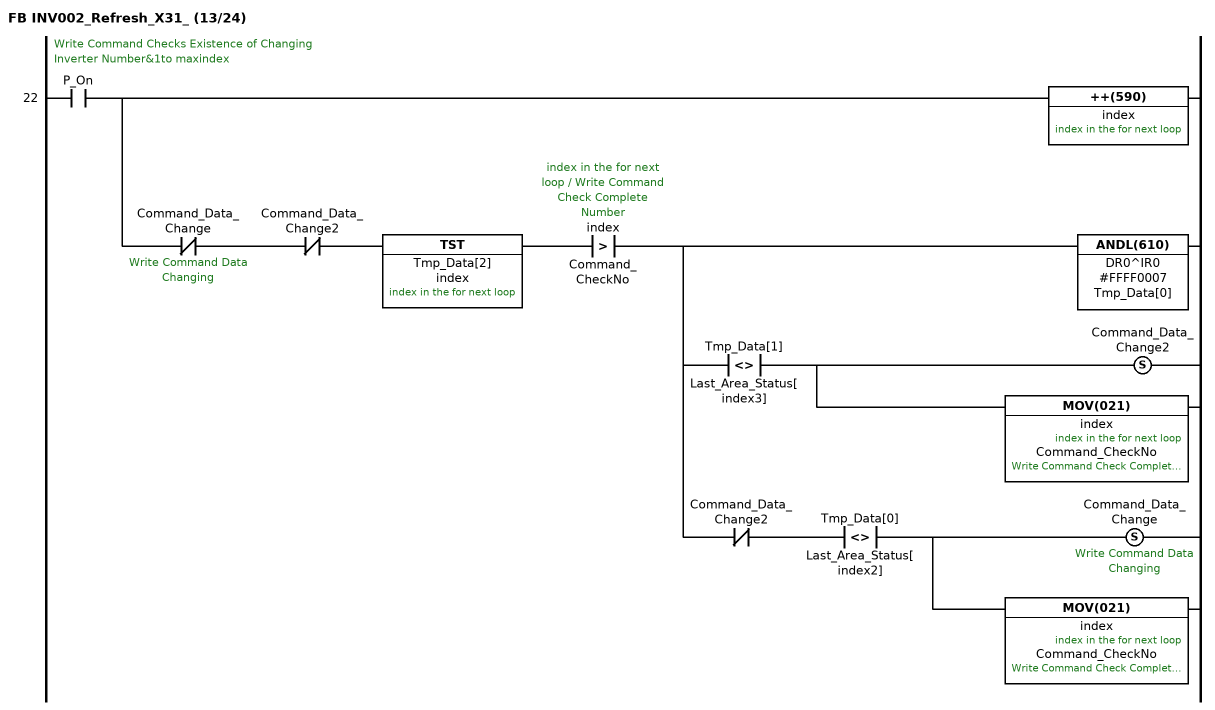
; [picture p24: FB INV002_Refresh_X31_, rungs 22-22]
; rung 22: Write Command Checks Existence of Changing / Inverter Number&1to maxindex
LD P_On
++(590) index  ; index in the for next loop
ANDNOT Command_Data_Change  ; Write Command Data Changing
ANDNOT Command_Data_Change2
ANDTST(350) Tmp_Data[2] index  ; index in the for next loop
AND>(320) index Command_CheckNo  ; index in the for next loop, Write Command Check Complete Number
OUT TR0
ANDL(610) DR0^IR0 #FFFF0007 Tmp_Data[0]
AND<>(305) Tmp_Data[1] Last_Area_Status[index3]
SET Command_Data_Change2
MOV(021) index Command_CheckNo  ; index in the for next loop, Write Command Check Complete Number
LD TR0
ANDNOT Command_Data_Change2
AND<>(305) Tmp_Data[0] Last_Area_Status[index2]
SET Command_Data_Change  ; Write Command Data Changing
MOV(021) index Command_CheckNo  ; index in the for next loop, Write Command Check Complete Number

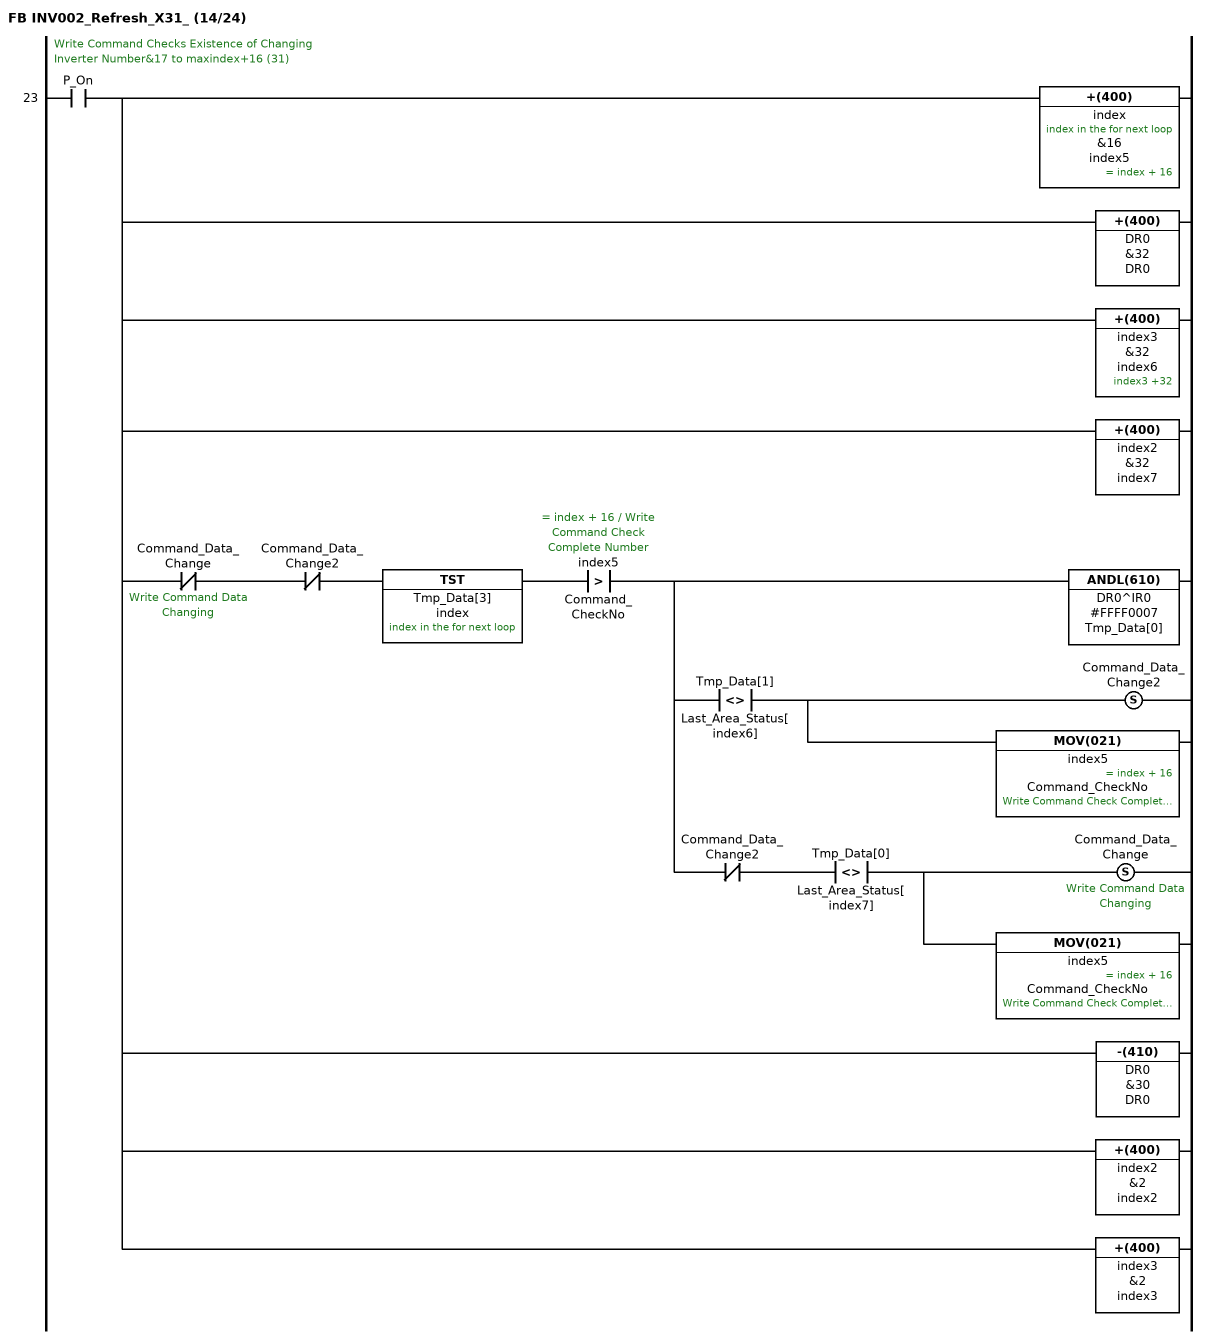
; rung 23: Write Command Checks Existence of Changing / Inverter Number&17 to maxindex+16 (31)
LD P_On
OUT TR0
+(400) index &16 index5  ; index in the for next loop, = index + 16
+(400) DR0 &32 DR0
+(400) index3 &32 index6  ; index3 +32
+(400) index2 &32 index7
ANDNOT Command_Data_Change  ; Write Command Data Changing
ANDNOT Command_Data_Change2
ANDTST(350) Tmp_Data[3] index  ; index in the for next loop
AND>(320) index5 Command_CheckNo  ; = index + 16, Write Command Check Complete Number
OUT TR1
ANDL(610) DR0^IR0 #FFFF0007 Tmp_Data[0]
AND<>(305) Tmp_Data[1] Last_Area_Status[index6]
SET Command_Data_Change2
MOV(021) index5 Command_CheckNo  ; = index + 16, Write Command Check Complete Number
LD TR1
ANDNOT Command_Data_Change2
AND<>(305) Tmp_Data[0] Last_Area_Status[index7]
SET Command_Data_Change  ; Write Command Data Changing
MOV(021) index5 Command_CheckNo  ; = index + 16, Write Command Check Complete Number
LD TR0
-(410) DR0 &30 DR0
+(400) index2 &2 index2
+(400) index3 &2 index3

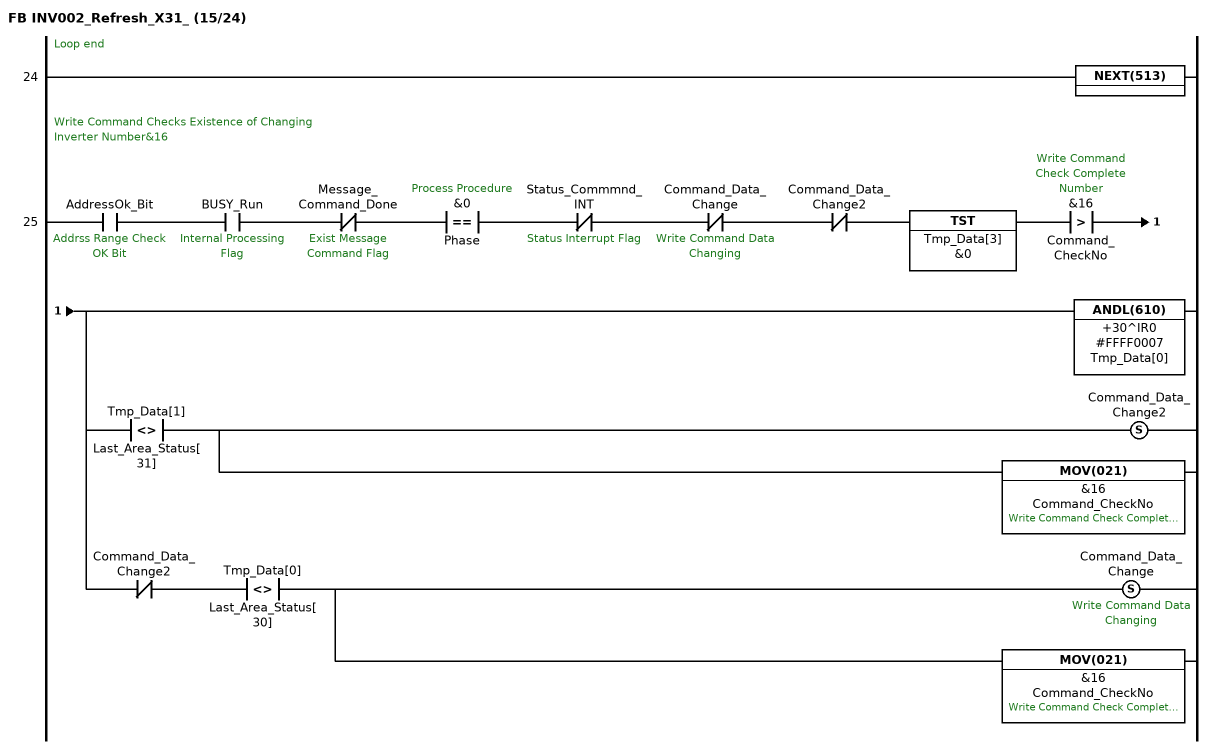
; rung 24: Loop end
NEXT(513)
; rung 25: Write Command Checks Existence of Changing / Inverter Number&16
LD AddressOk_Bit  ; Addrss Range Check OK Bit
AND BUSY_Run  ; Internal Processing Flag
ANDNOT Message_Command_Done  ; Exist Message Command Flag
AND=(300) &0 Phase  ; Process Procedure
ANDNOT Status_Commmnd_INT  ; Status Interrupt Flag
ANDNOT Command_Data_Change  ; Write Command Data Changing
ANDNOT Command_Data_Change2
ANDTST(350) Tmp_Data[3] &0
AND>(320) &16 Command_CheckNo  ; Write Command Check Complete Number
OUT TR0
ANDL(610) +30^IR0 #FFFF0007 Tmp_Data[0]
AND<>(305) Tmp_Data[1] Last_Area_Status[31]
SET Command_Data_Change2
MOV(021) &16 Command_CheckNo  ; Write Command Check Complete Number
LD TR0
ANDNOT Command_Data_Change2
AND<>(305) Tmp_Data[0] Last_Area_Status[30]
SET Command_Data_Change  ; Write Command Data Changing
MOV(021) &16 Command_CheckNo  ; Write Command Check Complete Number

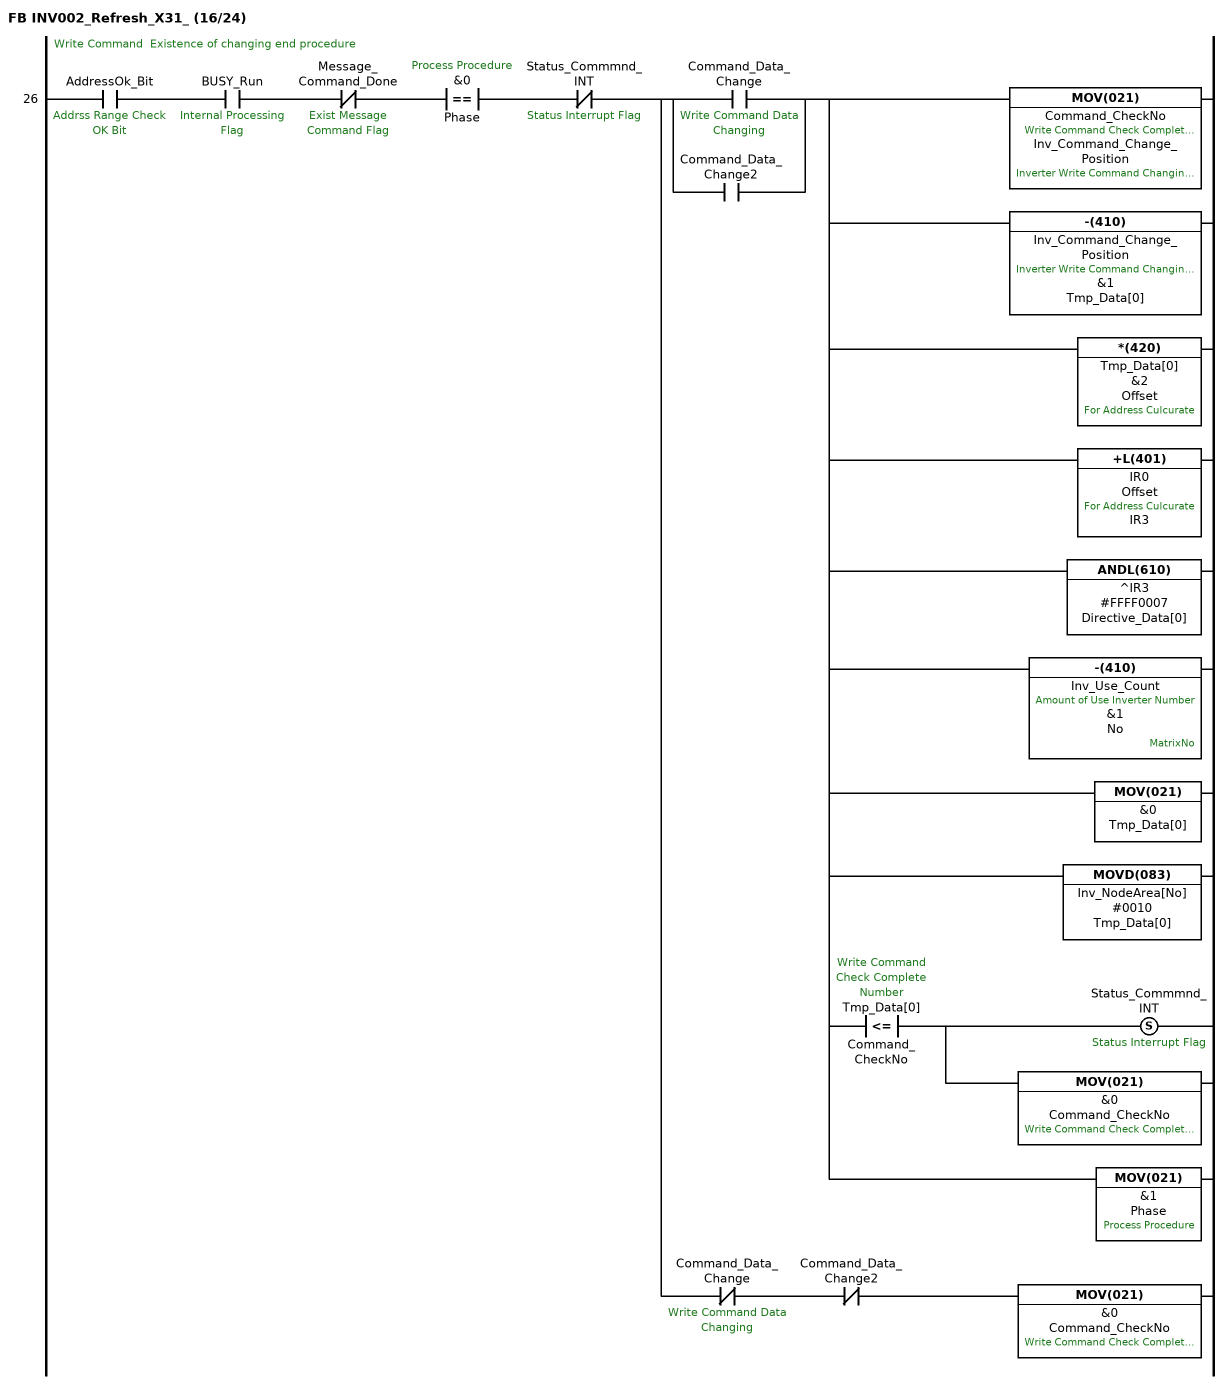
; rung 26: Write Command  Existence of changing end procedure
LD AddressOk_Bit  ; Addrss Range Check OK Bit
AND BUSY_Run  ; Internal Processing Flag
ANDNOT Message_Command_Done  ; Exist Message Command Flag
AND=(300) &0 Phase  ; Process Procedure
ANDNOT Status_Commmnd_INT  ; Status Interrupt Flag
OUT TR0
LD Command_Data_Change  ; Write Command Data Changing
OR Command_Data_Change2
ANDLD
OUT TR1
MOV(021) Command_CheckNo Inv_Command_Change_Position  ; Write Command Check Complete Number, Inverter Write Command Changing Position
-(410) Inv_Command_Change_Position &1 Tmp_Data[0]  ; Inverter Write Command Changing Position
*(420) Tmp_Data[0] &2 Offset  ; For Address Culcurate
+L(401) IR0 Offset IR3  ; For Address Culcurate
ANDL(610) ^IR3 #FFFF0007 Directive_Data[0]
-(410) Inv_Use_Count &1 No  ; Amount of Use Inverter Number, MatrixNo
MOV(021) &0 Tmp_Data[0]
MOVD(083) Inv_NodeArea[No] #0010 Tmp_Data[0]
AND<=(315) Tmp_Data[0] Command_CheckNo  ; Write Command Check Complete Number
SET Status_Commmnd_INT  ; Status Interrupt Flag
MOV(021) &0 Command_CheckNo  ; Write Command Check Complete Number
LD TR1
MOV(021) &1 Phase  ; Process Procedure
LD TR0
ANDNOT Command_Data_Change  ; Write Command Data Changing
ANDNOT Command_Data_Change2
MOV(021) &0 Command_CheckNo  ; Write Command Check Complete Number

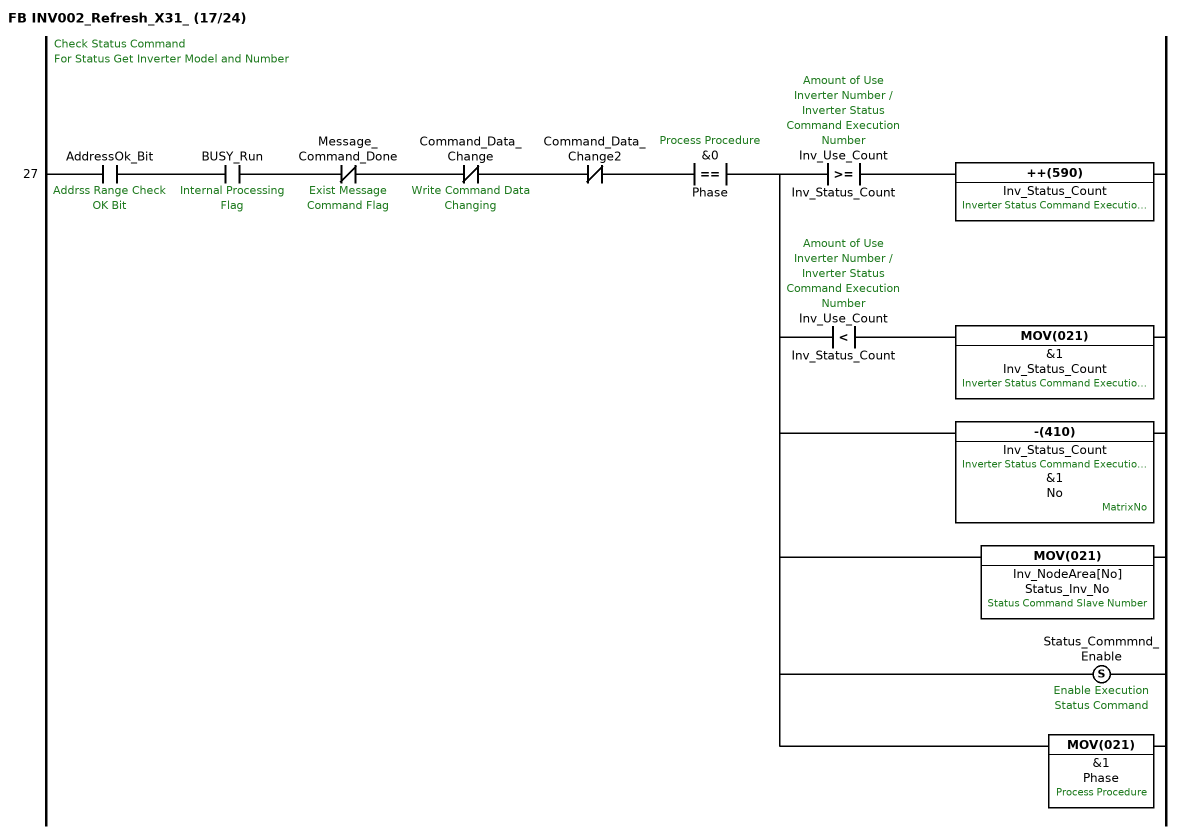
; rung 27: Check Status Command / For Status Get Inverter Model and Number
LD AddressOk_Bit  ; Addrss Range Check OK Bit
AND BUSY_Run  ; Internal Processing Flag
ANDNOT Message_Command_Done  ; Exist Message Command Flag
ANDNOT Command_Data_Change  ; Write Command Data Changing
ANDNOT Command_Data_Change2
AND=(300) &0 Phase  ; Process Procedure
OUT TR0
AND>=(325) Inv_Use_Count Inv_Status_Count  ; Amount of Use Inverter Number, Inverter Status Command Execution Number
++(590) Inv_Status_Count  ; Inverter Status Command Execution Number
LD TR0
AND<(310) Inv_Use_Count Inv_Status_Count  ; Amount of Use Inverter Number, Inverter Status Command Execution Number
MOV(021) &1 Inv_Status_Count  ; Inverter Status Command Execution Number
LD TR0
-(410) Inv_Status_Count &1 No  ; Inverter Status Command Execution Number, MatrixNo
MOV(021) Inv_NodeArea[No] Status_Inv_No  ; Status Command Slave Number
SET Status_Commmnd_Enable  ; Enable Execution Status Command
MOV(021) &1 Phase  ; Process Procedure

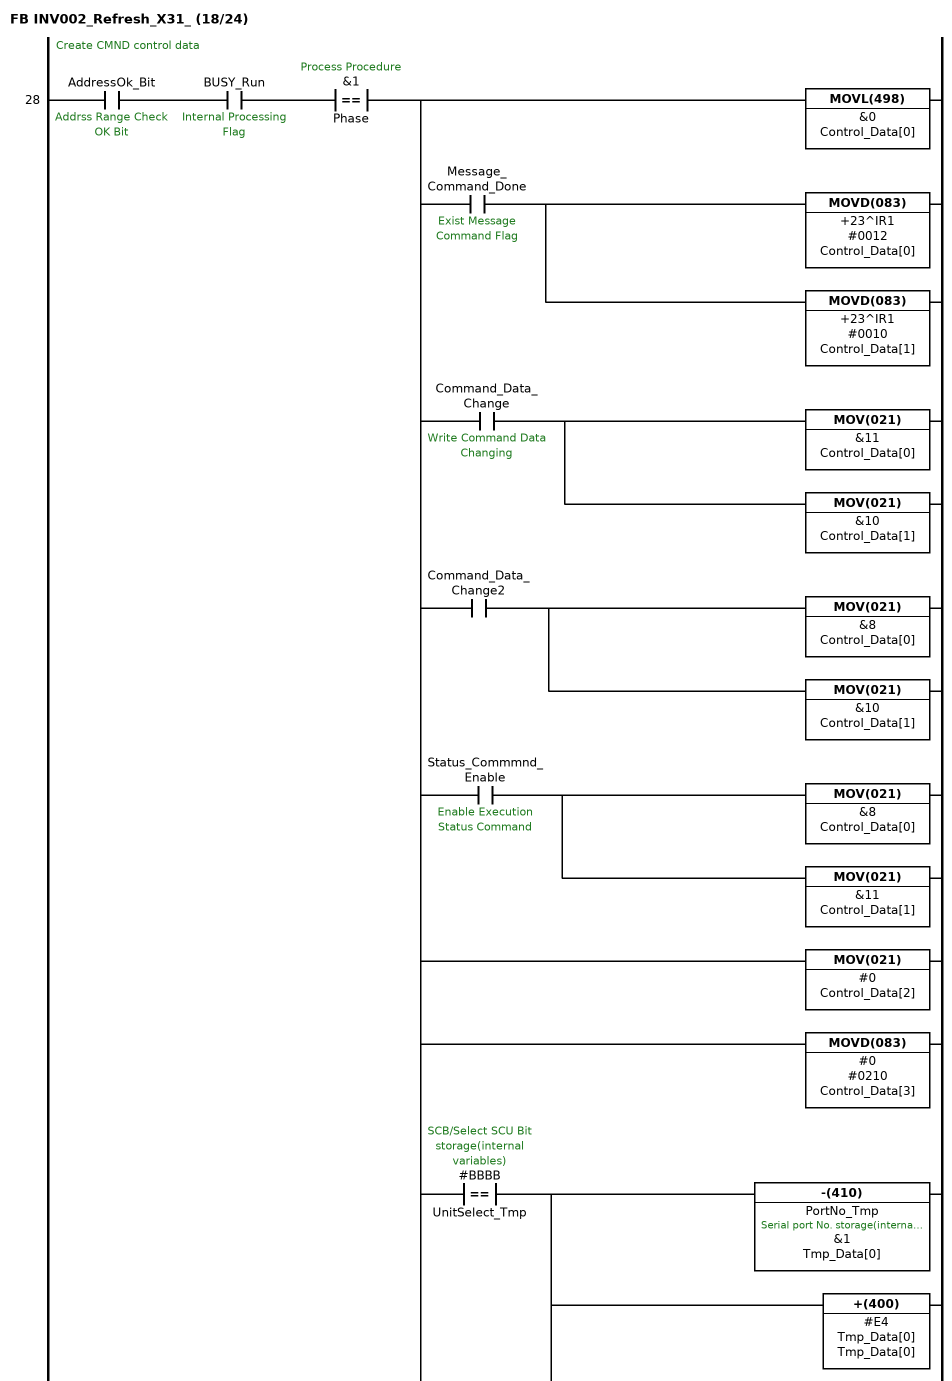

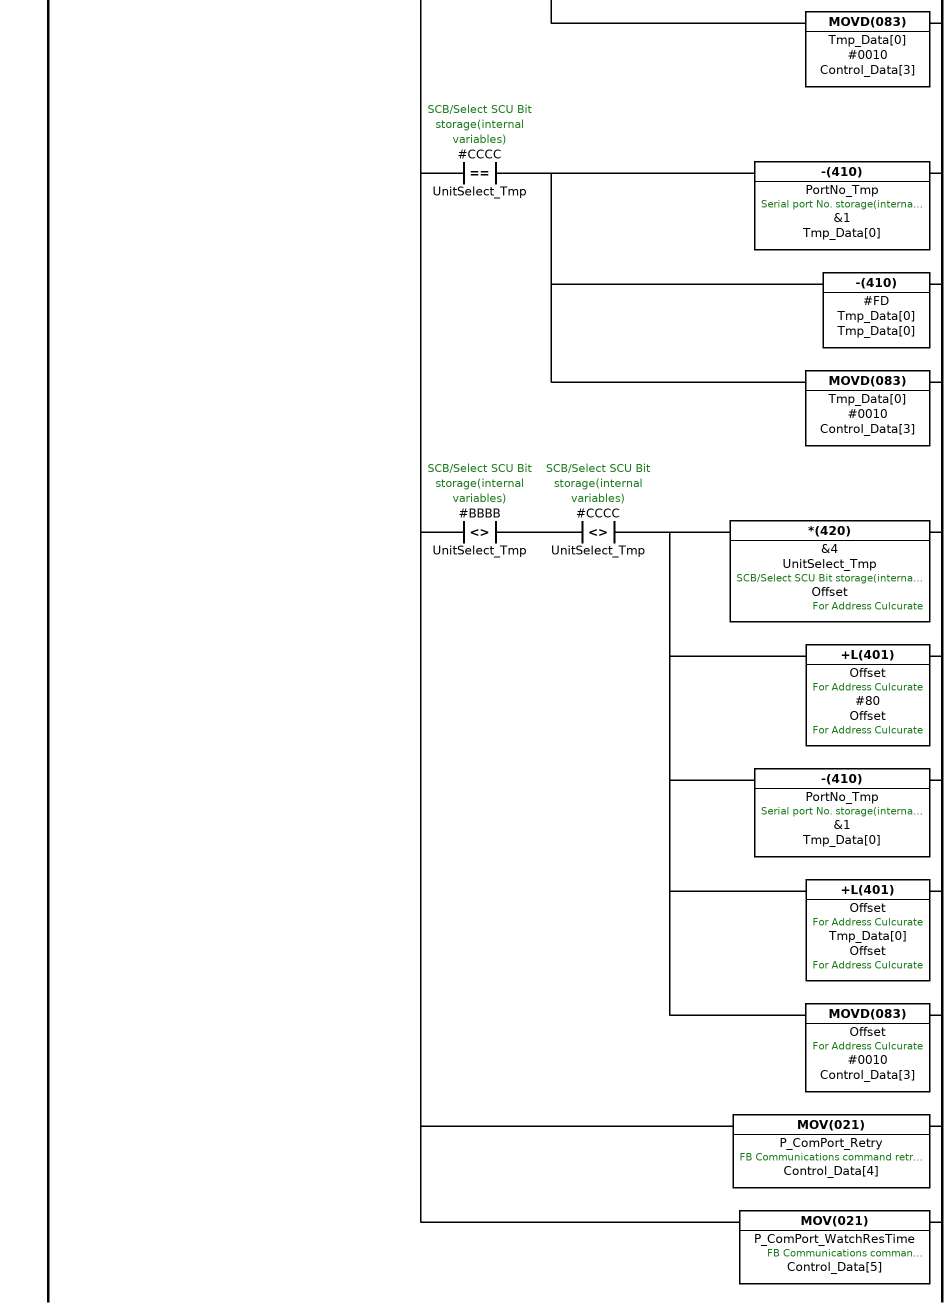
; rung 28: Create CMND control data
LD AddressOk_Bit  ; Addrss Range Check OK Bit
AND BUSY_Run  ; Internal Processing Flag
AND=(300) &1 Phase  ; Process Procedure
OUT TR0
MOVL(498) &0 Control_Data[0]
AND Message_Command_Done  ; Exist Message Command Flag
MOVD(083) +23^IR1 #0012 Control_Data[0]
MOVD(083) +23^IR1 #0010 Control_Data[1]
LD TR0
AND Command_Data_Change  ; Write Command Data Changing
MOV(021) &11 Control_Data[0]
MOV(021) &10 Control_Data[1]
LD TR0
AND Command_Data_Change2
MOV(021) &8 Control_Data[0]
MOV(021) &10 Control_Data[1]
LD TR0
AND Status_Commmnd_Enable  ; Enable Execution Status Command
MOV(021) &8 Control_Data[0]
MOV(021) &11 Control_Data[1]
LD TR0
MOV(021) #0 Control_Data[2]
MOVD(083) #0 #0210 Control_Data[3]
AND=(300) #BBBB UnitSelect_Tmp  ; SCB/Select SCU Bit storage(internal variables)
-(410) PortNo_Tmp &1 Tmp_Data[0]  ; Serial port No. storage(internal variables)
+(400) #E4 Tmp_Data[0] Tmp_Data[0]
MOVD(083) Tmp_Data[0] #0010 Control_Data[3]
LD TR0
AND=(300) #CCCC UnitSelect_Tmp  ; SCB/Select SCU Bit storage(internal variables)
-(410) PortNo_Tmp &1 Tmp_Data[0]  ; Serial port No. storage(internal variables)
-(410) #FD Tmp_Data[0] Tmp_Data[0]
MOVD(083) Tmp_Data[0] #0010 Control_Data[3]
LD TR0
AND<>(305) #BBBB UnitSelect_Tmp  ; SCB/Select SCU Bit storage(internal variables)
AND<>(305) #CCCC UnitSelect_Tmp  ; SCB/Select SCU Bit storage(internal variables)
*(420) &4 UnitSelect_Tmp Offset  ; SCB/Select SCU Bit storage(internal variables), For Address Culcurate
+L(401) Offset #80 Offset  ; For Address Culcurate
-(410) PortNo_Tmp &1 Tmp_Data[0]  ; Serial port No. storage(internal variables)
+L(401) Offset Tmp_Data[0] Offset  ; For Address Culcurate
MOVD(083) Offset #0010 Control_Data[3]  ; For Address Culcurate
LD TR0
MOV(021) P_ComPort_Retry Control_Data[4]  ; FB Communications command retry count
MOV(021) P_ComPort_WatchResTime Control_Data[5]  ; FB Communications command response Monitor time

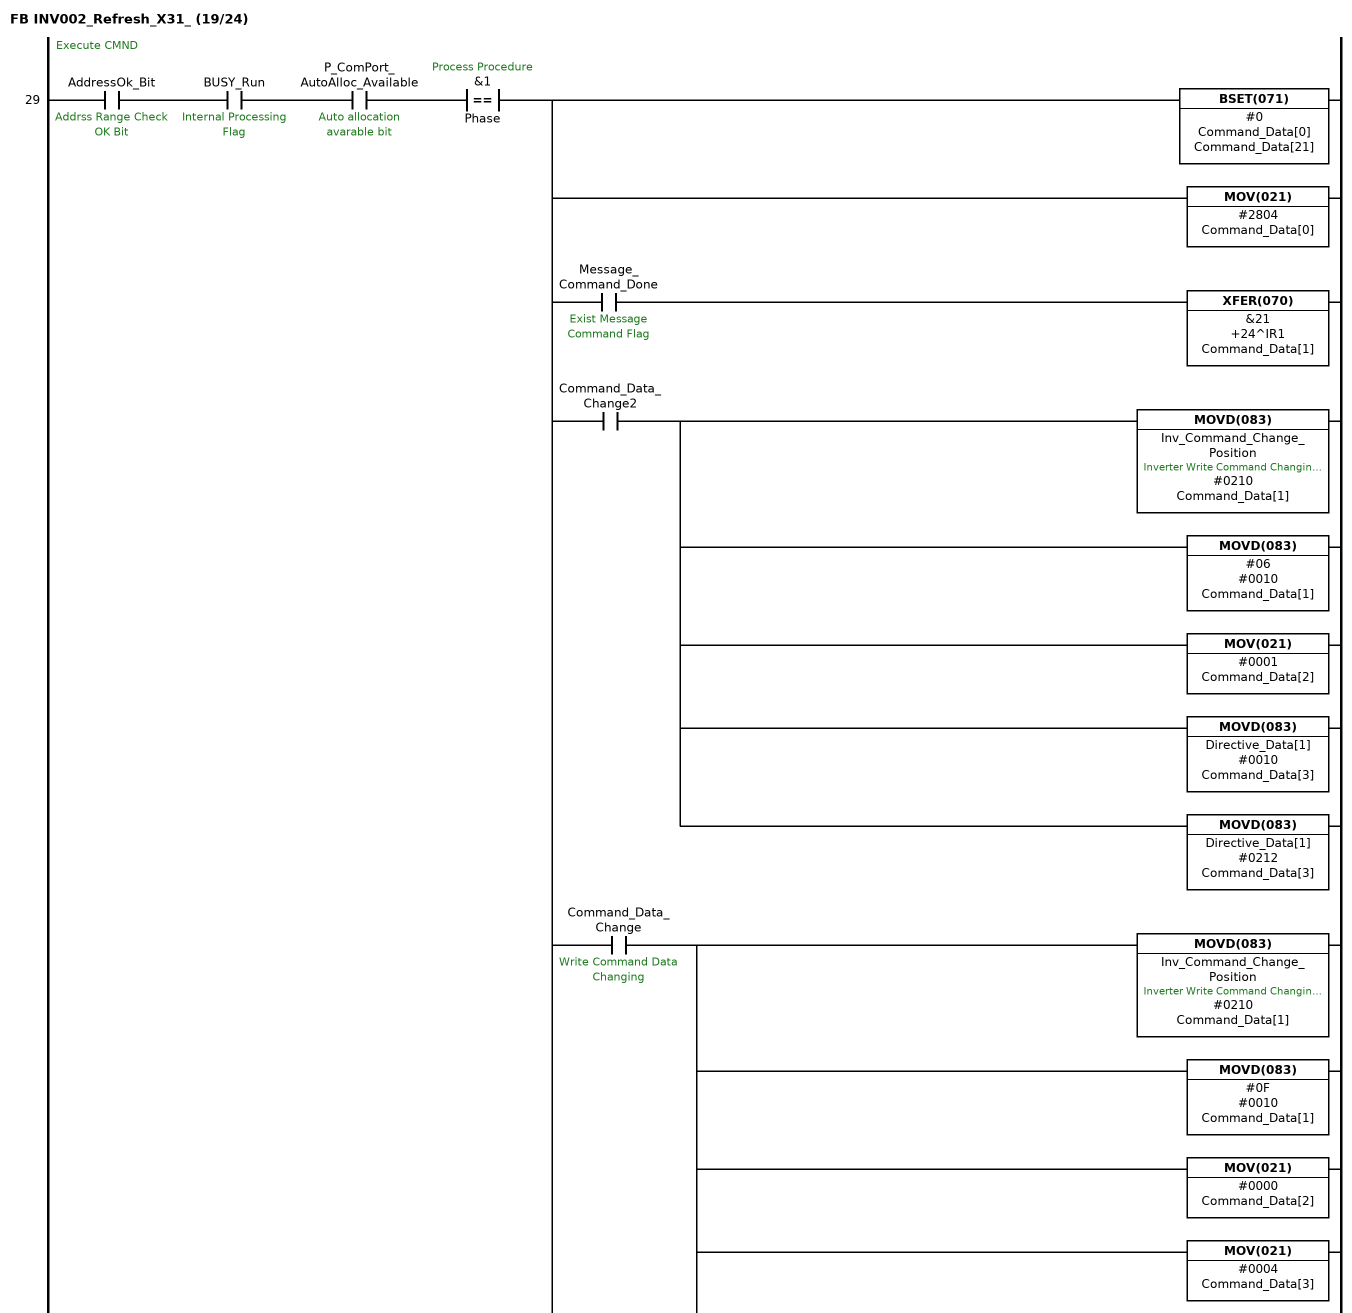

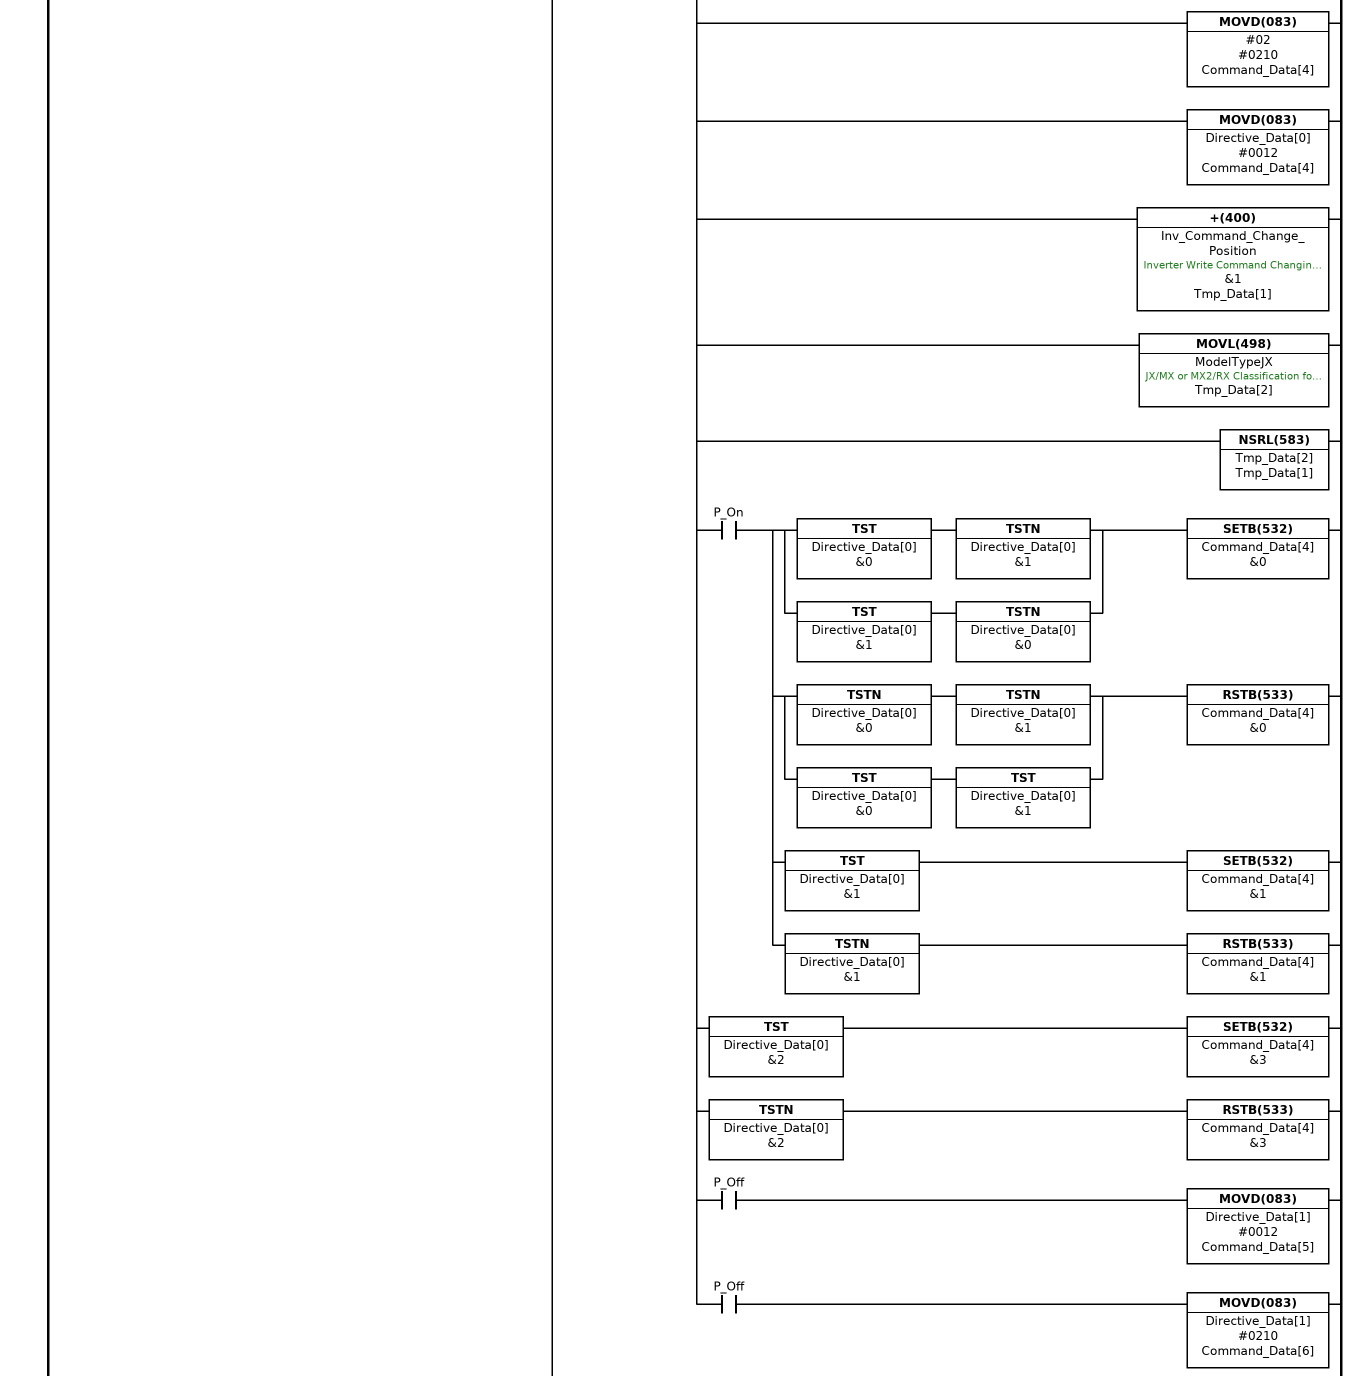

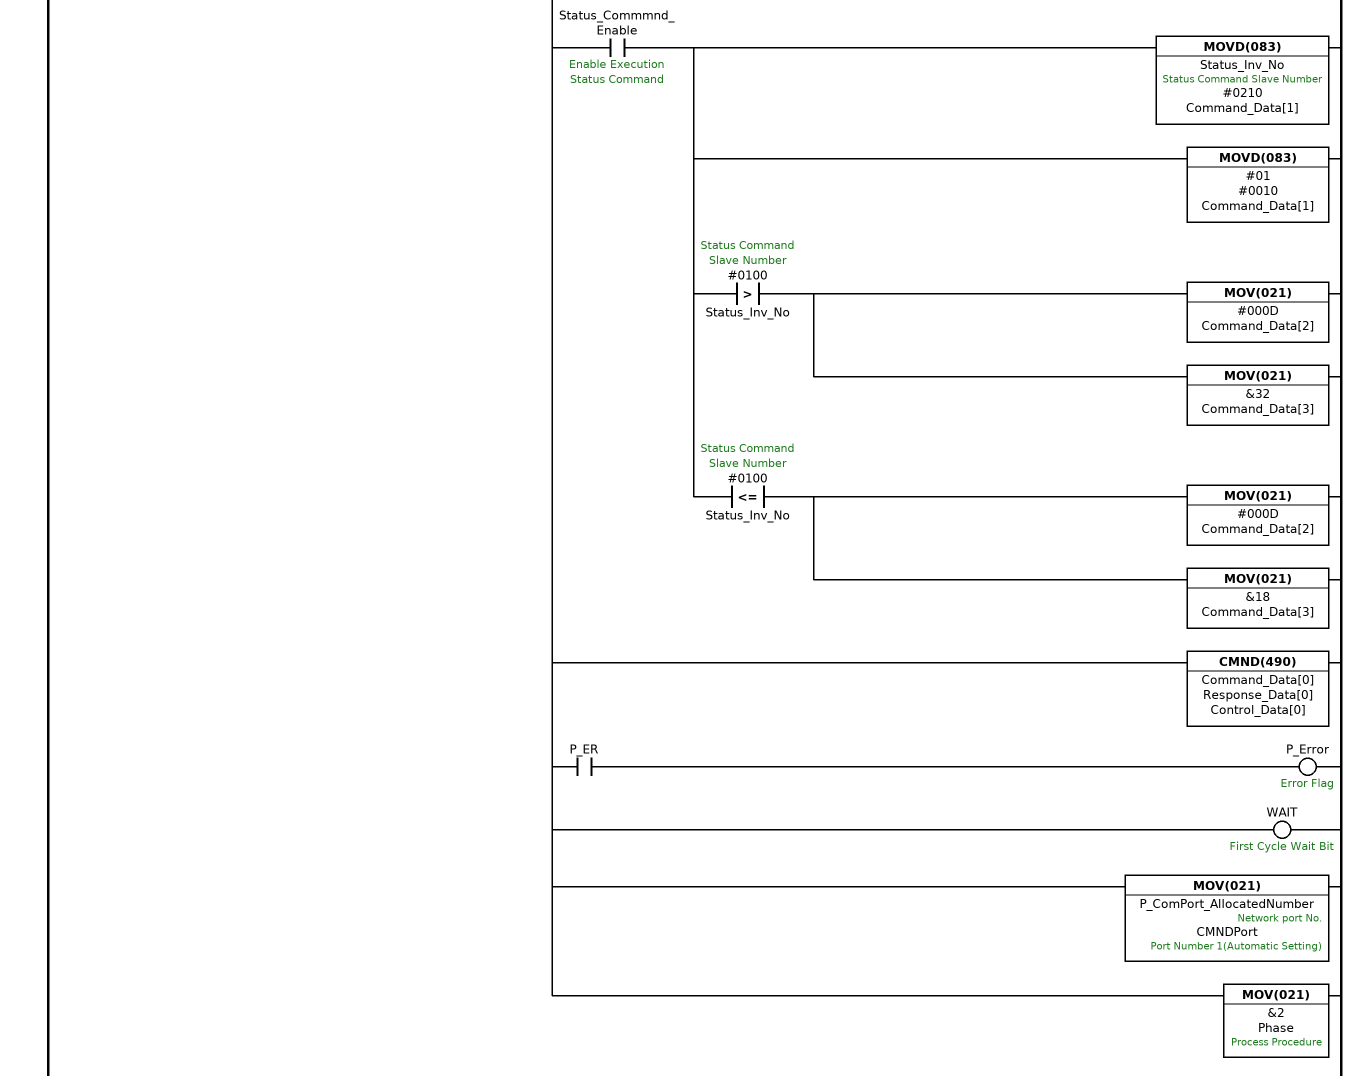
; rung 29: Execute CMND
LD AddressOk_Bit  ; Addrss Range Check OK Bit
AND BUSY_Run  ; Internal Processing Flag
AND P_ComPort_AutoAlloc_Available  ; Auto allocation avarable bit
AND=(300) &1 Phase  ; Process Procedure
OUT TR0
BSET(071) #0 Command_Data[0] Command_Data[21]
MOV(021) #2804 Command_Data[0]
AND Message_Command_Done  ; Exist Message Command Flag
XFER(070) &21 +24^IR1 Command_Data[1]
LD TR0
AND Command_Data_Change2
MOVD(083) Inv_Command_Change_Position #0210 Command_Data[1]  ; Inverter Write Command Changing Position
MOVD(083) #06 #0010 Command_Data[1]
MOV(021) #0001 Command_Data[2]
MOVD(083) Directive_Data[1] #0010 Command_Data[3]
MOVD(083) Directive_Data[1] #0212 Command_Data[3]
LD TR0
AND Command_Data_Change  ; Write Command Data Changing
OUT TR1
MOVD(083) Inv_Command_Change_Position #0210 Command_Data[1]  ; Inverter Write Command Changing Position
MOVD(083) #0F #0010 Command_Data[1]
MOV(021) #0000 Command_Data[2]
MOV(021) #0004 Command_Data[3]
MOVD(083) #02 #0210 Command_Data[4]
MOVD(083) Directive_Data[0] #0012 Command_Data[4]
+(400) Inv_Command_Change_Position &1 Tmp_Data[1]  ; Inverter Write Command Changing Position
MOVL(498) ModelTypeJX Tmp_Data[2]  ; JX/MX or MX2/RX Classification for older Inverter types also this Bit has to be set, like scanlist
NSRL(583) Tmp_Data[2] Tmp_Data[1]
AND P_On
OUT TR2
LDTST(350) Directive_Data[0] &0
ANDTSTN(351) Directive_Data[0] &1
LDTST(350) Directive_Data[0] &1
ANDTSTN(351) Directive_Data[0] &0
ORLD
ANDLD
SETB(532) Command_Data[4] &0
LD TR2
LDTSTN(351) Directive_Data[0] &0
ANDTSTN(351) Directive_Data[0] &1
LDTST(350) Directive_Data[0] &0
ANDTST(350) Directive_Data[0] &1
ORLD
ANDLD
RSTB(533) Command_Data[4] &0
LD TR2
ANDTST(350) Directive_Data[0] &1
SETB(532) Command_Data[4] &1
LD TR2
ANDTSTN(351) Directive_Data[0] &1
RSTB(533) Command_Data[4] &1
LD TR1
ANDTST(350) Directive_Data[0] &2
SETB(532) Command_Data[4] &3
LD TR1
ANDTSTN(351) Directive_Data[0] &2
RSTB(533) Command_Data[4] &3
LD TR1
AND P_Off
MOVD(083) Directive_Data[1] #0012 Command_Data[5]
LD TR1
AND P_Off
MOVD(083) Directive_Data[1] #0210 Command_Data[6]
LD TR0
AND Status_Commmnd_Enable  ; Enable Execution Status Command
OUT TR3
MOVD(083) Status_Inv_No #0210 Command_Data[1]  ; Status Command Slave Number
MOVD(083) #01 #0010 Command_Data[1]
AND>(320) #0100 Status_Inv_No  ; Status Command Slave Number
MOV(021) #000D Command_Data[2]
MOV(021) &32 Command_Data[3]
LD TR3
AND<=(315) #0100 Status_Inv_No  ; Status Command Slave Number
MOV(021) #000D Command_Data[2]
MOV(021) &18 Command_Data[3]
LD TR0
CMND(490) Command_Data[0] Response_Data[0] Control_Data[0]
AND P_ER
OUT P_Error  ; Error Flag
LD TR0
OUT WAIT  ; First Cycle Wait Bit
MOV(021) P_ComPort_AllocatedNumber CMNDPort  ; Network port No., Port Number 1(Automatic Setting)
MOV(021) &2 Phase  ; Process Procedure

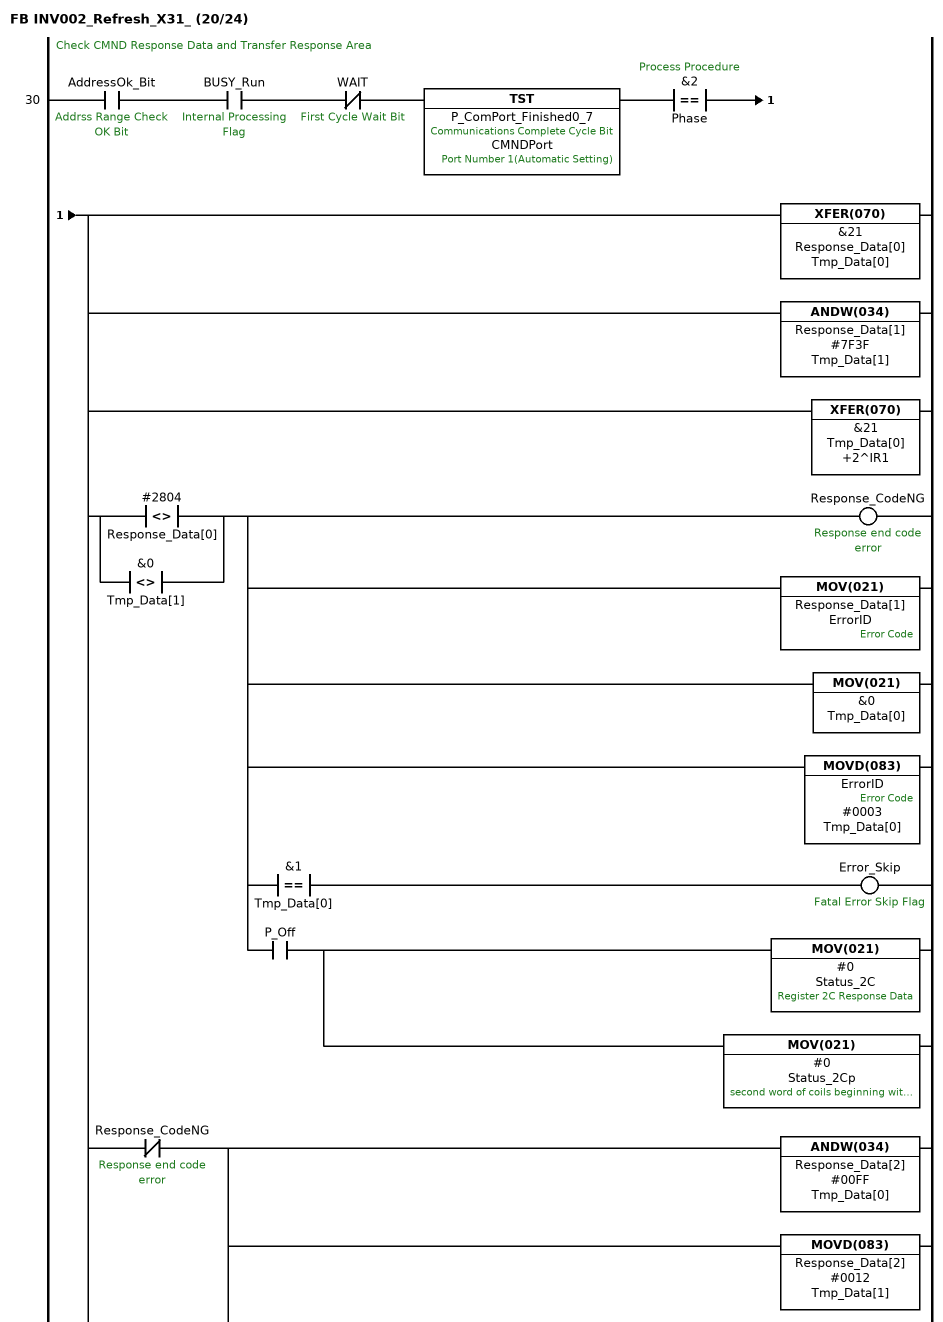

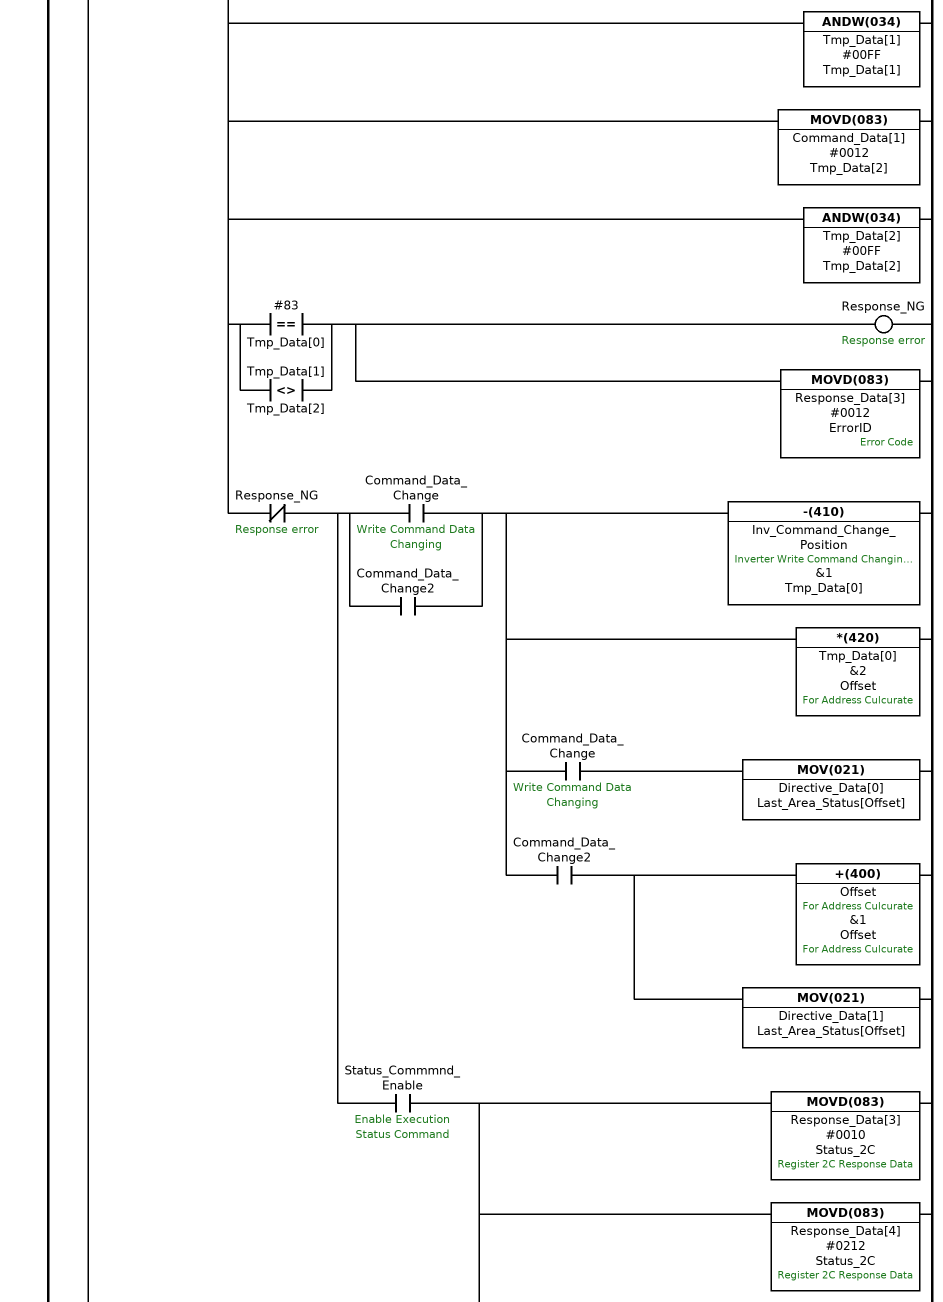

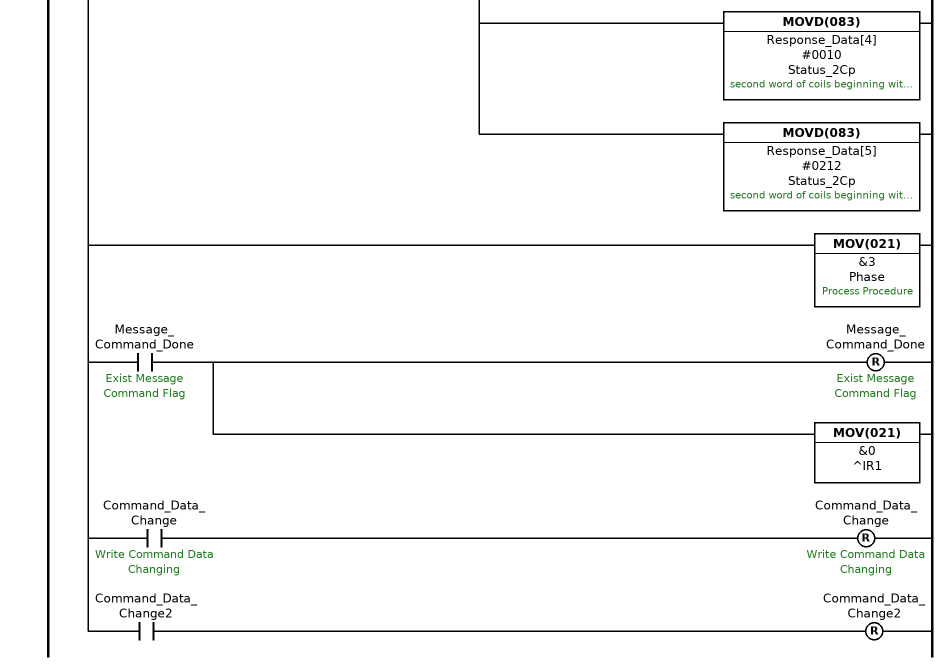
; rung 30: Check CMND Response Data and Transfer Response Area
LD AddressOk_Bit  ; Addrss Range Check OK Bit
AND BUSY_Run  ; Internal Processing Flag
ANDNOT WAIT  ; First Cycle Wait Bit
ANDTST(350) P_ComPort_Finished0_7 CMNDPort  ; Communications Complete Cycle Bit, Port Number 1(Automatic Setting)
AND=(300) &2 Phase  ; Process Procedure
OUT TR0
XFER(070) &21 Response_Data[0] Tmp_Data[0]
ANDW(034) Response_Data[1] #7F3F Tmp_Data[1]
XFER(070) &21 Tmp_Data[0] +2^IR1
LD<>(305) #2804 Response_Data[0]
OR<>(305) &0 Tmp_Data[1]
ANDLD
OUT TR1
OUT Response_CodeNG  ; Response end code error
MOV(021) Response_Data[1] ErrorID  ; Error Code
MOV(021) &0 Tmp_Data[0]
MOVD(083) ErrorID #0003 Tmp_Data[0]  ; Error Code
AND=(300) &1 Tmp_Data[0]
OUT Error_Skip  ; Fatal Error Skip Flag
LD TR1
AND P_Off
MOV(021) #0 Status_2C  ; Register 2C Response Data
MOV(021) #0 Status_2Cp  ; second word of coils beginning with coil 1F to 2E
LD TR0
ANDNOT Response_CodeNG  ; Response end code error
OUT TR2
ANDW(034) Response_Data[2] #00FF Tmp_Data[0]
MOVD(083) Response_Data[2] #0012 Tmp_Data[1]
ANDW(034) Tmp_Data[1] #00FF Tmp_Data[1]
MOVD(083) Command_Data[1] #0012 Tmp_Data[2]
ANDW(034) Tmp_Data[2] #00FF Tmp_Data[2]
LD=(300) #83 Tmp_Data[0]
OR<>(305) Tmp_Data[1] Tmp_Data[2]
ANDLD
OUT Response_NG  ; Response error
MOVD(083) Response_Data[3] #0012 ErrorID  ; Error Code
LD TR2
ANDNOT Response_NG  ; Response error
OUT TR3
LD Command_Data_Change  ; Write Command Data Changing
OR Command_Data_Change2
ANDLD
OUT TR4
-(410) Inv_Command_Change_Position &1 Tmp_Data[0]  ; Inverter Write Command Changing Position
*(420) Tmp_Data[0] &2 Offset  ; For Address Culcurate
AND Command_Data_Change  ; Write Command Data Changing
MOV(021) Directive_Data[0] Last_Area_Status[Offset]
LD TR4
AND Command_Data_Change2
+(400) Offset &1 Offset  ; For Address Culcurate
MOV(021) Directive_Data[1] Last_Area_Status[Offset]
LD TR3
AND Status_Commmnd_Enable  ; Enable Execution Status Command
MOVD(083) Response_Data[3] #0010 Status_2C  ; Register 2C Response Data
MOVD(083) Response_Data[4] #0212 Status_2C  ; Register 2C Response Data
MOVD(083) Response_Data[4] #0010 Status_2Cp  ; second word of coils beginning with coil 1F to 2E
MOVD(083) Response_Data[5] #0212 Status_2Cp  ; second word of coils beginning with coil 1F to 2E
LD TR0
MOV(021) &3 Phase  ; Process Procedure
AND Message_Command_Done  ; Exist Message Command Flag
RSET Message_Command_Done  ; Exist Message Command Flag
MOV(021) &0 ^IR1
LD TR0
AND Command_Data_Change  ; Write Command Data Changing
RSET Command_Data_Change  ; Write Command Data Changing
LD TR0
AND Command_Data_Change2
RSET Command_Data_Change2

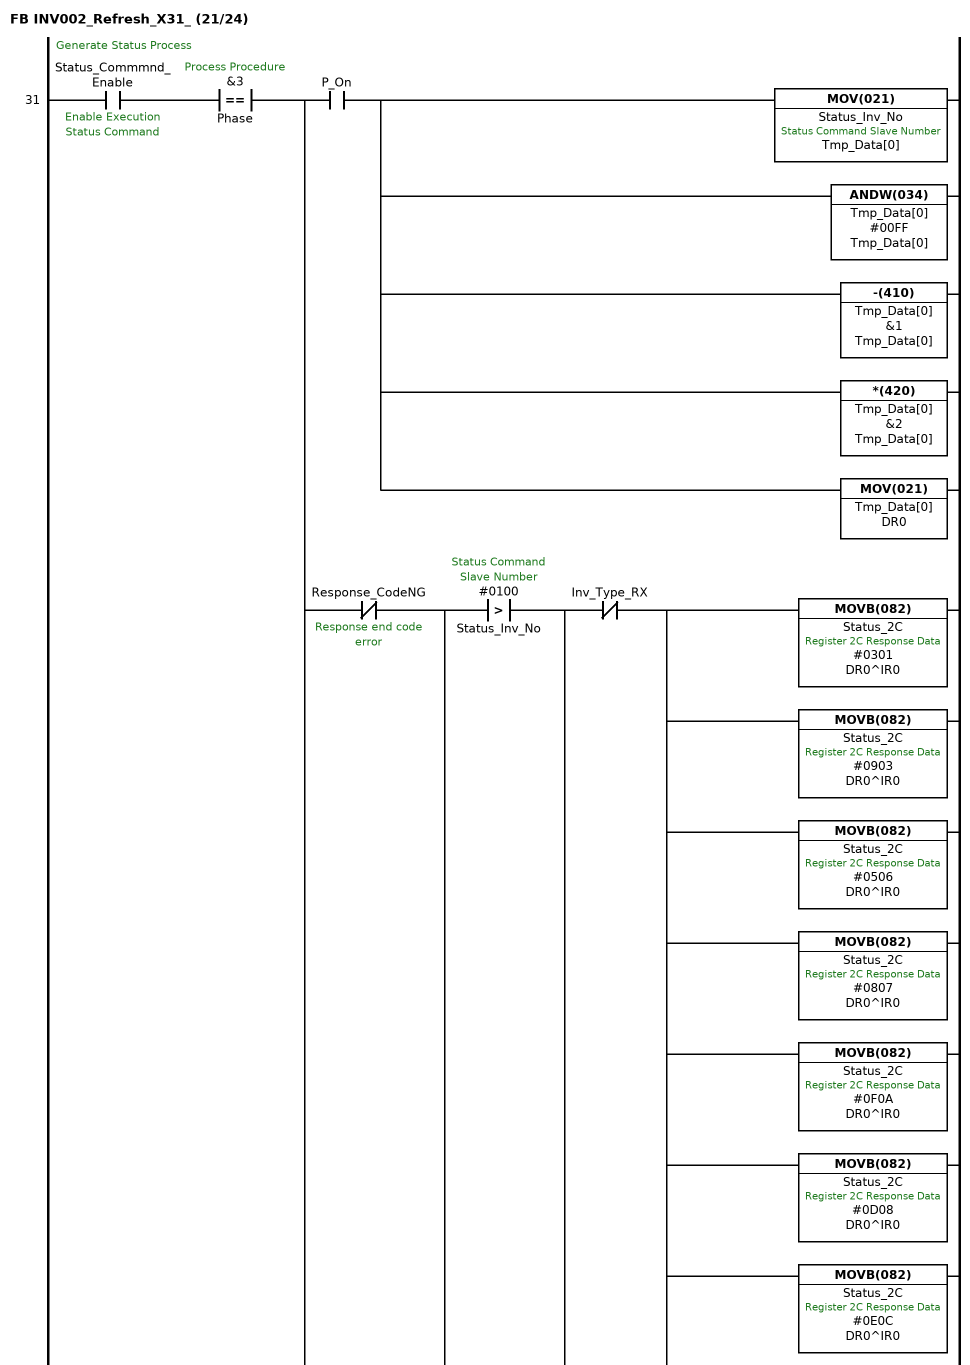

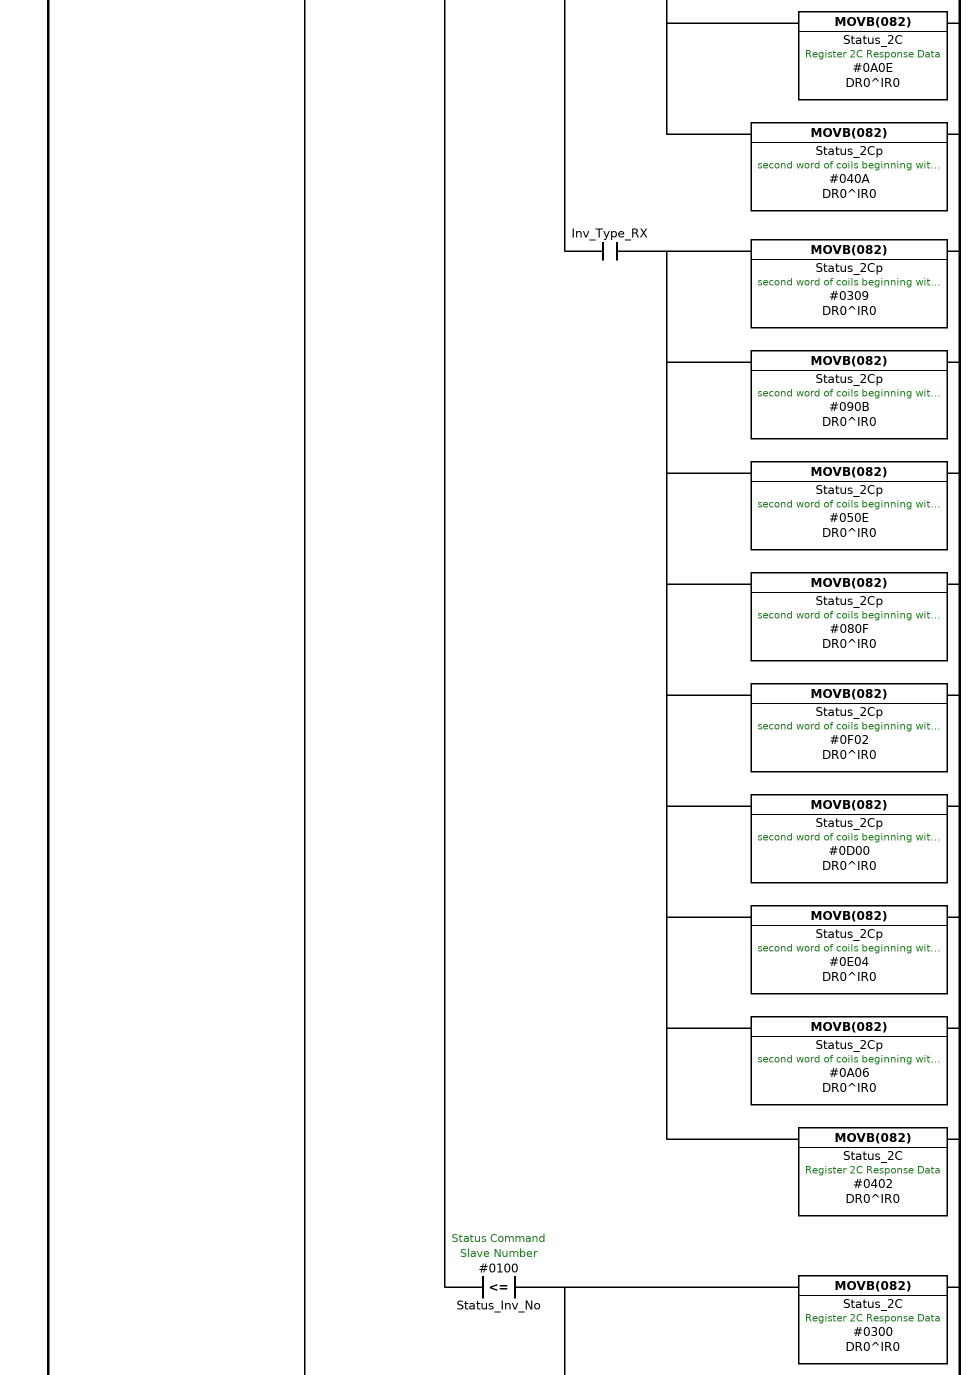

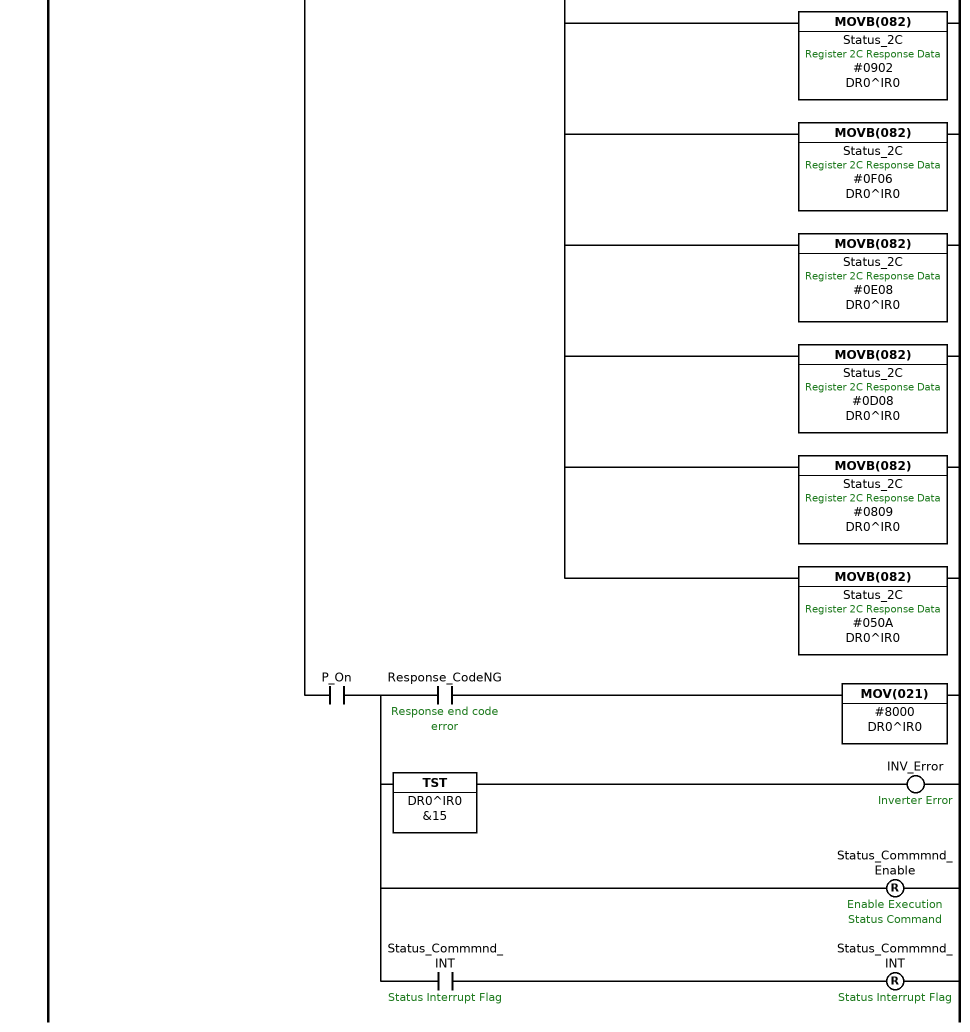
; rung 31: Generate Status Process
LD Status_Commmnd_Enable  ; Enable Execution Status Command
AND=(300) &3 Phase  ; Process Procedure
OUT TR0
AND P_On
MOV(021) Status_Inv_No Tmp_Data[0]  ; Status Command Slave Number
ANDW(034) Tmp_Data[0] #00FF Tmp_Data[0]
-(410) Tmp_Data[0] &1 Tmp_Data[0]
*(420) Tmp_Data[0] &2 Tmp_Data[0]
MOV(021) Tmp_Data[0] DR0
LD TR0
ANDNOT Response_CodeNG  ; Response end code error
OUT TR1
AND>(320) #0100 Status_Inv_No  ; Status Command Slave Number
OUT TR2
ANDNOT Inv_Type_RX
MOVB(082) Status_2C #0301 DR0^IR0  ; Register 2C Response Data
MOVB(082) Status_2C #0903 DR0^IR0  ; Register 2C Response Data
MOVB(082) Status_2C #0506 DR0^IR0  ; Register 2C Response Data
MOVB(082) Status_2C #0807 DR0^IR0  ; Register 2C Response Data
MOVB(082) Status_2C #0F0A DR0^IR0  ; Register 2C Response Data
MOVB(082) Status_2C #0D08 DR0^IR0  ; Register 2C Response Data
MOVB(082) Status_2C #0E0C DR0^IR0  ; Register 2C Response Data
MOVB(082) Status_2C #0A0E DR0^IR0  ; Register 2C Response Data
MOVB(082) Status_2Cp #040A DR0^IR0  ; second word of coils beginning with coil 1F to 2E
LD TR2
AND Inv_Type_RX
MOVB(082) Status_2Cp #0309 DR0^IR0  ; second word of coils beginning with coil 1F to 2E
MOVB(082) Status_2Cp #090B DR0^IR0  ; second word of coils beginning with coil 1F to 2E
MOVB(082) Status_2Cp #050E DR0^IR0  ; second word of coils beginning with coil 1F to 2E
MOVB(082) Status_2Cp #080F DR0^IR0  ; second word of coils beginning with coil 1F to 2E
MOVB(082) Status_2Cp #0F02 DR0^IR0  ; second word of coils beginning with coil 1F to 2E
MOVB(082) Status_2Cp #0D00 DR0^IR0  ; second word of coils beginning with coil 1F to 2E
MOVB(082) Status_2Cp #0E04 DR0^IR0  ; second word of coils beginning with coil 1F to 2E
MOVB(082) Status_2Cp #0A06 DR0^IR0  ; second word of coils beginning with coil 1F to 2E
MOVB(082) Status_2C #0402 DR0^IR0  ; Register 2C Response Data
LD TR1
AND<=(315) #0100 Status_Inv_No  ; Status Command Slave Number
MOVB(082) Status_2C #0300 DR0^IR0  ; Register 2C Response Data
MOVB(082) Status_2C #0902 DR0^IR0  ; Register 2C Response Data
MOVB(082) Status_2C #0F06 DR0^IR0  ; Register 2C Response Data
MOVB(082) Status_2C #0E08 DR0^IR0  ; Register 2C Response Data
MOVB(082) Status_2C #0D08 DR0^IR0  ; Register 2C Response Data
MOVB(082) Status_2C #0809 DR0^IR0  ; Register 2C Response Data
MOVB(082) Status_2C #050A DR0^IR0  ; Register 2C Response Data
LD TR0
AND P_On
OUT TR3
AND Response_CodeNG  ; Response end code error
MOV(021) #8000 DR0^IR0
LD TR3
ANDTST(350) DR0^IR0 &15
OUT INV_Error  ; Inverter Error
LD TR3
RSET Status_Commmnd_Enable  ; Enable Execution Status Command
AND Status_Commmnd_INT  ; Status Interrupt Flag
RSET Status_Commmnd_INT  ; Status Interrupt Flag

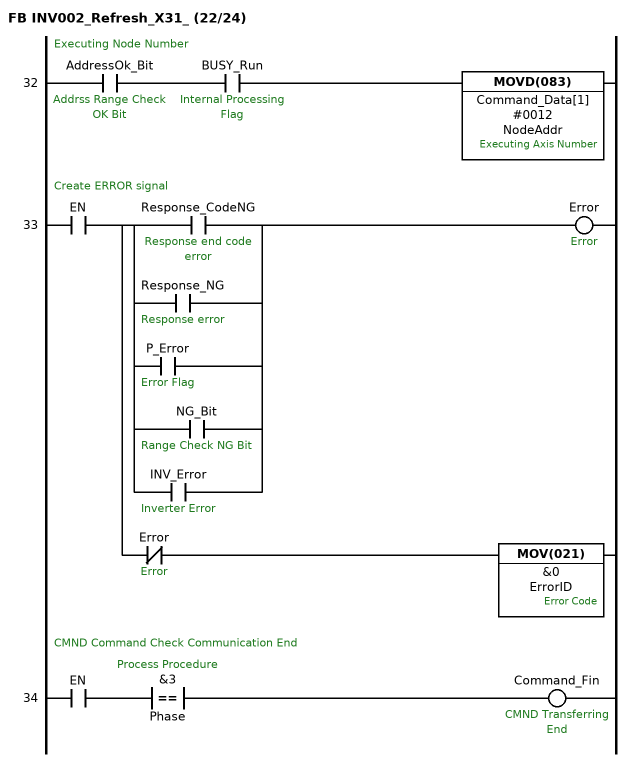
; rung 32: Executing Node Number
LD AddressOk_Bit  ; Addrss Range Check OK Bit
AND BUSY_Run  ; Internal Processing Flag
MOVD(083) Command_Data[1] #0012 NodeAddr  ; Executing Axis Number
; rung 33: Create ERROR signal
LD EN
OUT TR0
LD Response_CodeNG  ; Response end code error
OR Response_NG  ; Response error
OR P_Error  ; Error Flag
OR NG_Bit  ; Range Check NG Bit
OR INV_Error  ; Inverter Error
ANDLD
OUT Error  ; Error
LD TR0
ANDNOT Error  ; Error
MOV(021) &0 ErrorID  ; Error Code
; rung 34: CMND Command Check Communication End
LD EN
AND=(300) &3 Phase  ; Process Procedure
OUT Command_Fin  ; CMND Transferring End

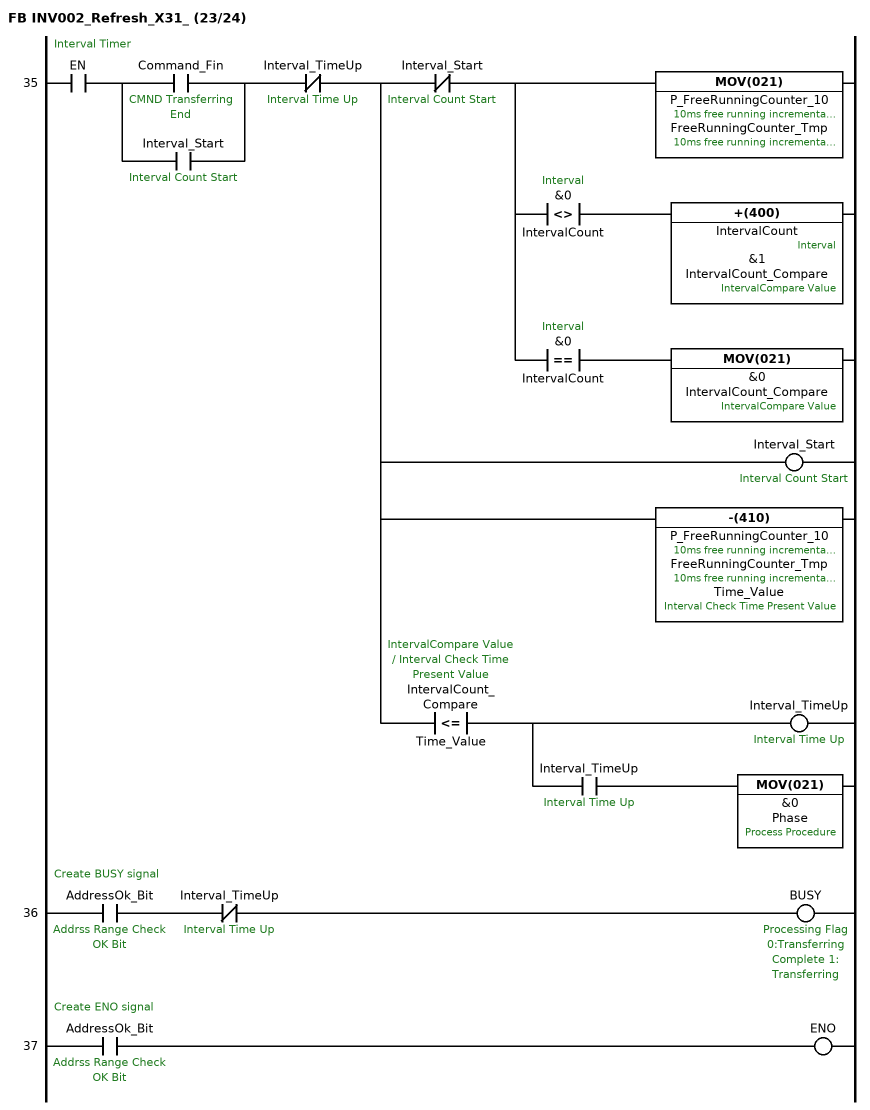
; rung 35: Interval Timer
LD EN
LD Command_Fin  ; CMND Transferring End
OR Interval_Start  ; Interval Count Start
ANDLD
ANDNOT Interval_TimeUp  ; Interval Time Up
OUT TR0
ANDNOT Interval_Start  ; Interval Count Start
OUT TR1
MOV(021) P_FreeRunningCounter_10 FreeRunningCounter_Tmp  ; 10ms free running incremental counter, 10ms free running incremental counter record
AND<>(305) &0 IntervalCount  ; Interval
+(400) IntervalCount &1 IntervalCount_Compare  ; Interval, IntervalCompare Value
LD TR1
AND=(300) &0 IntervalCount  ; Interval
MOV(021) &0 IntervalCount_Compare  ; IntervalCompare Value
LD TR0
OUT Interval_Start  ; Interval Count Start
-(410) P_FreeRunningCounter_10 FreeRunningCounter_Tmp Time_Value  ; 10ms free running incremental counter, 10ms free running incremental counter record, Interval Check Time Present Value
AND<=(315) IntervalCount_Compare Time_Value  ; IntervalCompare Value, Interval Check Time Present Value
OUT Interval_TimeUp  ; Interval Time Up
AND Interval_TimeUp  ; Interval Time Up
MOV(021) &0 Phase  ; Process Procedure
; rung 36: Create BUSY signal
LD AddressOk_Bit  ; Addrss Range Check OK Bit
ANDNOT Interval_TimeUp  ; Interval Time Up
OUT BUSY  ; Processing Flag 0:Transferring Complete 1:Transferring
; rung 37: Create ENO signal
LD AddressOk_Bit  ; Addrss Range Check OK Bit
OUT ENO

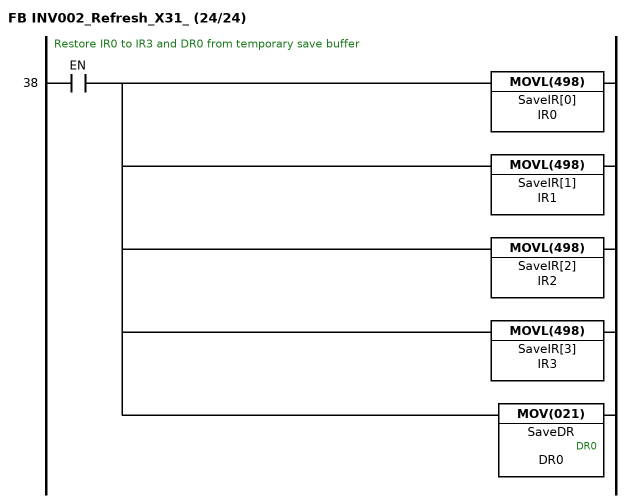
; rung 38: Restore IR0 to IR3 and DR0 from temporary save buffer
LD EN
MOVL(498) SaveIR[0] IR0
MOVL(498) SaveIR[1] IR1
MOVL(498) SaveIR[2] IR2
MOVL(498) SaveIR[3] IR3
MOV(021) SaveDR DR0  ; DR0